// TwinCAT 3 PLC project SCADA_V2
// ProgramVersion: 3.1.4024.0
// libraries:
//   PlantControl and CMs, * (ArmAutomation)
//   Tc2_ControllerToolbox, * (Beckhoff Automation GmbH)
//   Tc2_Standard, * (Beckhoff Automation GmbH)
//   Tc2_System, * (Beckhoff Automation GmbH)
//   Tc3_Module, * (Beckhoff Automation GmbH)
// project tree:
//   GVLs/ CMD.TcGVL, HMI.TcGVL, GVL.TcGVL, PAR.TcGVL, SEQ.TcGVL, SIM.TcGVL
//   / PlcTask.TcTTO
//   POUs/CMs/ CM_AI_CALL.TcPOU, CM_DO_3state_CALL.TcPOU, CM_DO_CALL.TcPOU
//   POUs/EQ Modules/ EQ_CALL.TcPOU, EQ_Conveyor_V1.TcPOU
//   POUs/HVAC/ HVAC_B28_CM_CALL.TcPOU, HVAC_B28_Main_Seq.TcPOU
//   POUs/Plant Control/ FB_PlantControl_B57.TcPOU, FB_PlantControl_B28.TcPOU
//   POUs/Regulators/ PRG_FB_CTRL_PID.TcPOU, PRG_PID_CALL.TcPOU
//   POUs/ SITE_100MS.TcPOU, SITE_MAIN_CYCLIC.TcPOU
//   POUs/Simulations/ CALL_SIM.TcPOU, FBALT_2_PUMPS_GRAPH.TcPOU, FB_ALT_2_PUMPS.TcPOU, SIM_Analog_Input.TcPOU, SIM_Valve_Damper_OPEN_CLOSE.TcPOU
// real-time tasks:
//   TASK SITE_MAIN_CYCLIC: cycle T#10ms, priority 20, ADS port 350
//   TASK SITE_100MS: cycle T#100000us, priority 1, ADS port 351

CONFIGURATION SCADA_V2
    RESOURCE PLC ON TwinCAT3
        TASK PlcTask(INTERVAL := T#10ms, PRIORITY := 20);
        PROGRAM SITE_MAIN_CYCLIC WITH PlcTask : SITE_MAIN_CYCLIC;
        PROGRAM SITE_100MS WITH PlcTask : SITE_100MS;
    END_RESOURCE
END_CONFIGURATION

// ---- GVLs/CMD.TcGVL
{attribute 'qualified_only'}
VAR_GLOBAL
	Plant_B57_Control : PlantAndCMs.Udt_PlantControl;
	
	Plant_B28_Control : PlantAndCMs.Udt_PlantControl;
END_VAR

// ---- GVLs/HMI.TcGVL
{attribute 'qualified_only'}
VAR_GLOBAL
	
	//CMs for HVAC
	CM_AV_1 : PlantAndCMs.Udt_CM_Actuator2State_V2;
	
	CM_PU_AO_1 : PlantAndCMs.Udt_CM_AO_V2;
	
	CM_MTR_AO_1 : PlantAndCMs.Udt_CM_AO_V2;
	MTR_1_PO_PV : DINT;
	
	CM_DMP_AO_1 : PlantAndCMs.Udt_CM_Actuator2State_V2;
	
	//CMs For EQs
	CM_MTR_3State : PlantAndCMs.Udt_CM_Actuator3State_V2;

	//
	outputFromPressure_1 : LREAL;
	
	
	//PID
	CM_DMP_1_PID_PARAMS : ST_CTRL_PID_PARAMS;
	CM_MTR_1_PID_PARAMS : ST_CTRL_PID_PARAMS;
	
	//Simulation parameters
	
	
	
	
	
	//SP
	
	MTR_1_MAN_SP : DINT;
	DMP_1_MAN_SP : DINT;
	
END_VAR

// ---- GVLs/GVL.TcGVL
{attribute 'qualified_only'}
VAR_GLOBAL
	
	mb_Input_Coils    :    ARRAY [0..255] OF BOOL;
	mb_Output_Coils :    ARRAY [0..255] OF BOOL;
	mb_Input_Registers :    ARRAY [0..255] OF WORD; // Modbus TCP master side function code = 04 (read only)
	mb_Output_Registers :    ARRAY [0..255] OF WORD; // Modbus TCP master side function code = 03 & 16 (read/write)
	 
END_VAR

// ---- GVLs/PAR.TcGVL
{attribute 'qualified_only'}
VAR_GLOBAL
	
	// DAMPER SP
	
	DMP_1_SP : INT; 
	
	//Motor SP
	
	MTR_1_SP : DINT;

END_VAR

// ---- GVLs/SEQ.TcGVL
{attribute 'qualified_only'}
VAR_GLOBAL
	
	// HVAC_SEQ_28
	
	B28_STEP_1: BOOL;
	B28_STEP_2 : BOOL;
	B28_STEP_3 : BOOL;
	B28_STEP_4 : BOOL;
	B28_STEP_5 : BOOL;
	B28_STEP_6: BOOL;

END_VAR

// ---- GVLs/SIM.TcGVL
{attribute 'qualified_only'}
VAR_GLOBAL
	
	Pressure_1_Input : DINT;
	Pressure_1 : REAL ;
	
	//Sim Damper
	
	Feedback_Open : BOOL;
	Feedback_Closed : BOOL;
	
	DMP_1_INPUT : DINT;
	DMP_1_OUTPUT : DINT;
	
	MTR_1_InputFromPID : DINT;
	MTR_1_OutputToPID : DINT;
	
	// Conveyor sim
	
	CV_ON: BOOL;
	CCV_ON: BOOL;
	
END_VAR

// ---- POUs/SITE_MAIN_CYCLIC.TcPOU
PROGRAM SITE_MAIN_CYCLIC
VAR
	PlantControl_B57 : FB_PlantControl_B57;
	PlantControl_B28 : FB_PlantControl_B28;
	
	SIM_CALL : CALL_SIM;
	
	HVAC_CM_CALL : HVAC_B28_CM_CALL;
	
	HVAC_MAIN_SEQ : HVAC_B28_Main_Seq;
	
	cm_AI_CALL : CM_AI_CALL;
	cm_DO_3State_CALL : CM_DO_3state_CALL;
	
END_VAR

PlantControl_B28();
PlantControl_B57();


//B28
HVAC_CM_CALL();
HVAC_MAIN_SEQ();

//For testing:
EQ_CALL();
SIM_CALL();

// CMs
cm_AI_CALL();
//cm_DO_3State_CALL();

END_PROGRAM

// ---- POUs/Plant Control/FB_PlantControl_B57.TcPOU
FUNCTION_BLOCK FB_PlantControl_B57

VAR
	Plant_Control : PlantAndCMs.FB_PlantControl_V2;
	
	
	MB_START : BOOL;
	MB_EMG_STOP : BOOL;
END_VAR

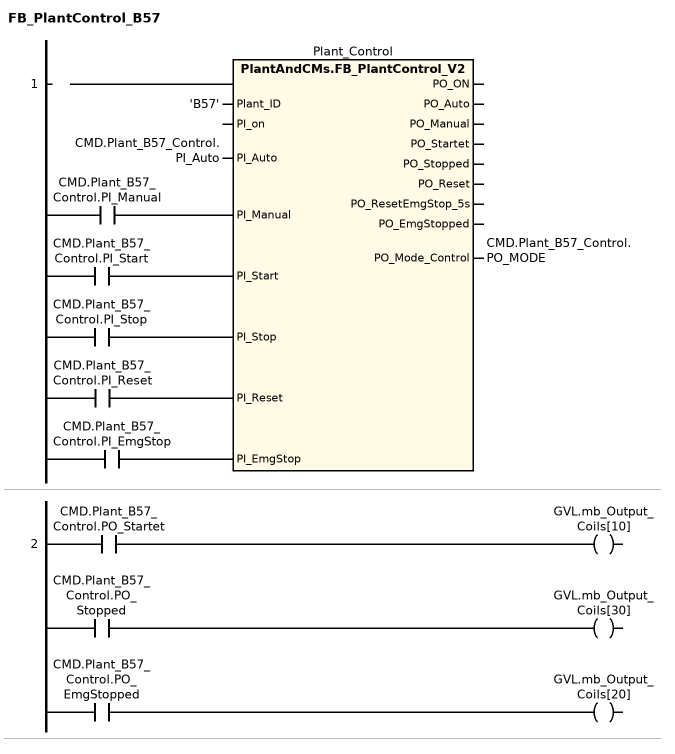
// NETWORK 1
Plant_Control(
    Plant_ID := 'B57',
    PI_Auto := CMD.Plant_B57_Control.PI_Auto,
    PI_Manual := CMD.Plant_B57_Control.PI_Manual,
    PI_Start := CMD.Plant_B57_Control.PI_Start,
    PI_Stop := CMD.Plant_B57_Control.PI_Stop,
    PI_Reset := CMD.Plant_B57_Control.PI_Reset,
    PI_EmgStop := CMD.Plant_B57_Control.PI_EmgStop,
    PO_Mode_Control => CMD.Plant_B57_Control.PO_MODE); // PlantAndCMs.FB_PlantControl_V2

// NETWORK 2
GVL.mb_Output_Coils[10] := CMD.Plant_B57_Control.PO_Startet;
GVL.mb_Output_Coils[30] := CMD.Plant_B57_Control.PO_Stopped;
GVL.mb_Output_Coils[20] := CMD.Plant_B57_Control.PO_EmgStopped;

END_FUNCTION_BLOCK

// ---- POUs/Plant Control/FB_PlantControl_B28.TcPOU
FUNCTION_BLOCK FB_PlantControl_B28

VAR
	Plant_Control : PlantAndCMs.FB_PlantControl_V2;
	
	
	MB_START : BOOL;
	MB_EMG_STOP : BOOL;
END_VAR

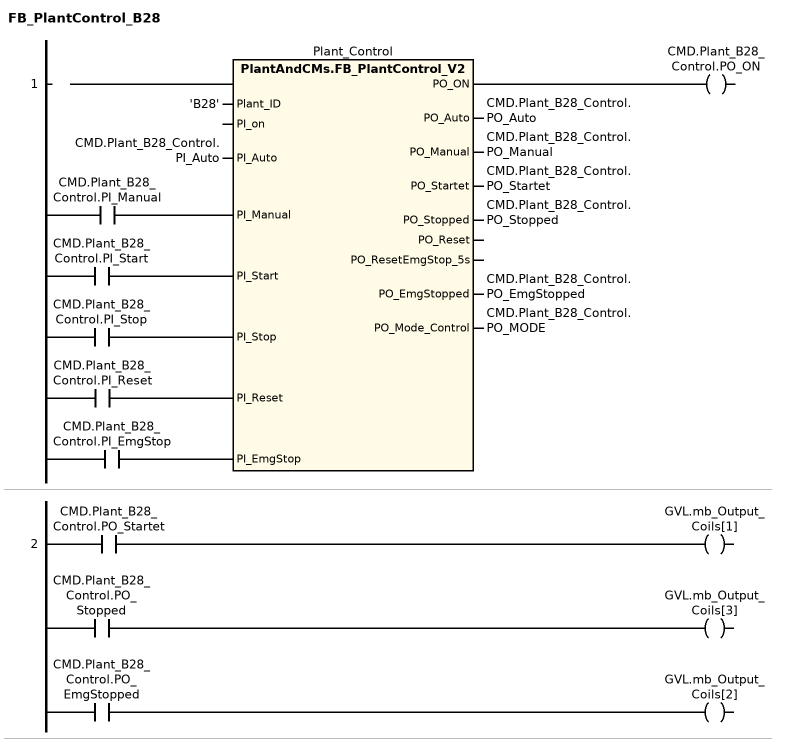
// NETWORK 1
Plant_Control(
    Plant_ID := 'B28',
    PI_Auto := CMD.Plant_B28_Control.PI_Auto,
    PI_Manual := CMD.Plant_B28_Control.PI_Manual,
    PI_Start := CMD.Plant_B28_Control.PI_Start,
    PI_Stop := CMD.Plant_B28_Control.PI_Stop,
    PI_Reset := CMD.Plant_B28_Control.PI_Reset,
    PI_EmgStop := CMD.Plant_B28_Control.PI_EmgStop,
    PO_Auto => CMD.Plant_B28_Control.PO_Auto,
    PO_Manual => CMD.Plant_B28_Control.PO_Manual,
    PO_Startet => CMD.Plant_B28_Control.PO_Startet,
    PO_Stopped => CMD.Plant_B28_Control.PO_Stopped,
    PO_EmgStopped => CMD.Plant_B28_Control.PO_EmgStopped,
    PO_Mode_Control => CMD.Plant_B28_Control.PO_MODE); // PlantAndCMs.FB_PlantControl_V2
CMD.Plant_B28_Control.PO_ON := Plant_Control.PO_ON;

// NETWORK 2
GVL.mb_Output_Coils[1] := CMD.Plant_B28_Control.PO_Startet;
GVL.mb_Output_Coils[3] := CMD.Plant_B28_Control.PO_Stopped;
GVL.mb_Output_Coils[2] := CMD.Plant_B28_Control.PO_EmgStopped;

END_FUNCTION_BLOCK

// ---- POUs/Simulations/CALL_SIM.TcPOU
FUNCTION_BLOCK CALL_SIM
VAR_INPUT
END_VAR
VAR_OUTPUT
END_VAR
VAR
	Damper_1_SIM : SIM_Valve_Damper_OPEN_CLOSE;
	
	pressure_1_SIM : SIM_Analog_Input;
	
	fb_ALT_2_PUMPS : FB_ALT_2_PUMPS;
	LS1:BOOL;
	LS2:BOOL;
	LS3:BOOL;
	LS4:BOOL;
	
	Pump_1 : BOOL;
	Pump_2 : BOOL;
	min_limit: INT;
END_VAR


IF SEQ.B28_STEP_2 THEN
	Damper_1_SIM(
	max_limit := PAR.DMP_1_SP,
	min_limit := 0,
	
	Start_Open := SEQ.B28_STEP_2,
	Start_Close := FALSE,//SEQ.B28_STEP_3,
	Open_Finish => SIM.Feedback_Open,
	Close_Finish => SIM.Feedback_Closed,
	open_status => SIM.DMP_1_OUTPUT
	
);
END_IF


fb_ALT_2_PUMPS(
	LS_1 := LS1,
	LS_2 := LS2,
	LS_3 := LS3,
	
	Pump_1 => Pump_1,
	Pump_2 => Pump_2
	);

pressure_1_SIM(
	EnableSim := CMD.Plant_B28_Control.PO_ON,
	AutoMode := SEQ.B28_STEP_3,
	ManualValue :=  HMI.MTR_1_MAN_SP,
	AutoSpeed := 0.1,
	MinValue := 15000,
	MaxValue := 30000,
	ManualValue := 10,
	SimulatedValue => SIM.Pressure_1,
	);

END_FUNCTION_BLOCK

// ---- POUs/Simulations/SIM_Valve_Damper_OPEN_CLOSE.TcPOU
FUNCTION_BLOCK SIM_Valve_Damper_OPEN_CLOSE
VAR_INPUT
    Start_Open  : BOOL;
    Start_Close : BOOL;
    max_limit   : INT;
    min_limit   : INT;
END_VAR

VAR_OUTPUT
    Open_Finish  : BOOL:= FALSE;
    Close_Finish : BOOL := FALSE;
    open_status  : INT := 0;
END_VAR

VAR
    timer : TON;
END_VAR

// Start timer only if movement is requested and not yet at limit
IF (Start_Open AND open_status < max_limit) OR (Start_Close AND open_status > min_limit) THEN
    timer(IN := TRUE, PT := T#1S);
ELSE
    timer(IN := FALSE);
END_IF

// On timer expiration, step open_status up or down
IF timer.Q THEN
    IF Start_Open AND open_status < max_limit THEN
        open_status := open_status + 1;
    ELSIF Start_Close AND open_status > min_limit THEN
        open_status := open_status - 1;
    END_IF
    timer(IN := FALSE); // Reset timer after action
END_IF

// Output flags
Open_Finish  := (open_status >= max_limit);
Close_Finish := (open_status <= min_limit);

END_FUNCTION_BLOCK

// ---- POUs/Simulations/SIM_Analog_Input.TcPOU
FUNCTION_BLOCK SIM_Analog_Input
VAR_INPUT
    EnableSim   : BOOL;
    AutoMode    : BOOL;
    ManualValue : REAL;
    AutoSpeed   : REAL;         // e.g. 0.1
    
	MinValue    : REAL;         // e.g. 0.0
    MaxValue    : REAL;         // e.g. 100.0
END_VAR

VAR_OUTPUT
    SimulatedValue : REAL;
END_VAR

VAR
    timeCounter : REAL := 0.0;
    timer       : TON;
END_VAR

// Auto simulation mode
IF EnableSim THEN
    IF AutoMode THEN
        timer(IN := TRUE, PT := T#500ms);
        IF timer.Q THEN
            timer(IN := FALSE); // reset
            timeCounter := timeCounter + AutoSpeed;
            SimulatedValue := (MaxValue - MinValue)/2.0 * SIN(timeCounter) + (MaxValue + MinValue)/2.0;
        END_IF
    ELSE
        // Manual override mode
        SimulatedValue := LIMIT(MinValue, ManualValue, MaxValue);
    END_IF
ELSE
    // Simulation disabled
    SimulatedValue := 0.0;
    timer(IN := FALSE);
END_IF

END_FUNCTION_BLOCK

// ---- POUs/Simulations/FB_ALT_2_PUMPS.TcPOU
FUNCTION_BLOCK FB_ALT_2_PUMPS
VAR_INPUT
	LS_1 : BOOL;
	LS_2 : BOOL;
	LS_3 : BOOL;
	LS_4 : BOOL;
END_VAR
VAR_OUTPUT
	Pump_1 : BOOL;
	Pump_2 : BOOL;
END_VAR
VAR
	Reset_pumps: BOOL;
	Alt_pumps: BOOL;
	
	Pump_Count : INT := 0;
	LS_2_Pump_1: BOOL;
	LS_2_Pump_2: BOOL;
	LS_3_Pump_1: BOOL;
	LS_3_Pump_2: BOOL;
END_VAR
VAR // added by the converter: edge detectors and wires of the graphical bodies
    _rt1 : R_TRIG;
    _w1, _w2, _w3 : BOOL;
END_VAR

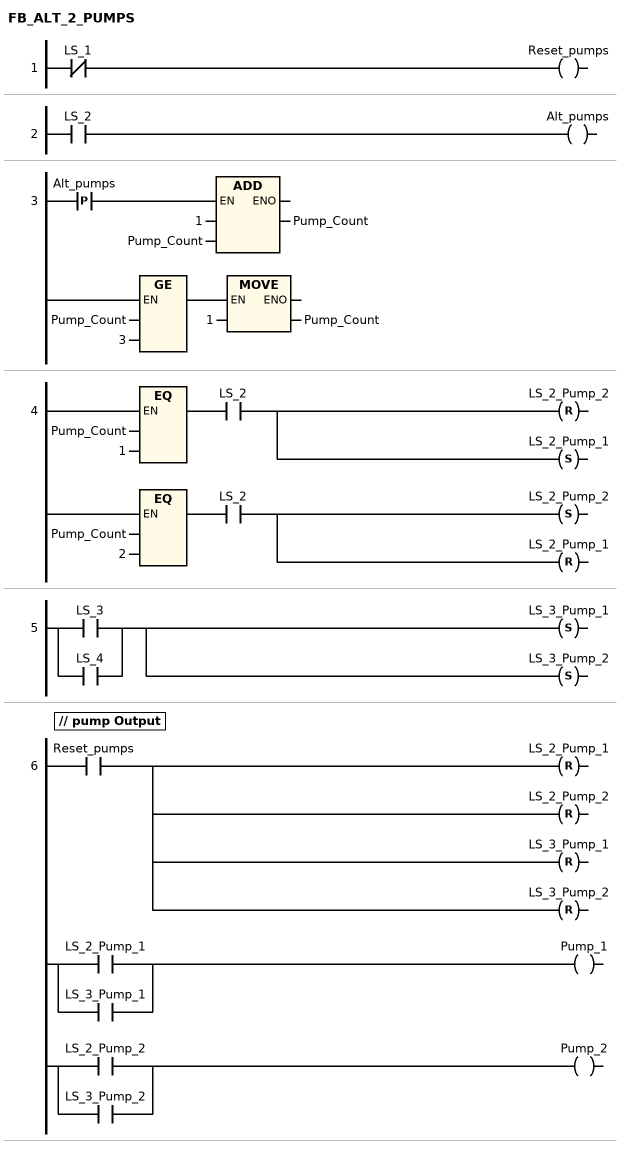
// NETWORK 1
Reset_pumps := NOT LS_1;

// NETWORK 2
Alt_pumps := LS_2;

// NETWORK 3
_rt1(CLK := Alt_pumps);
IF _rt1.Q THEN Pump_Count := 1 + Pump_Count; END_IF
IF Pump_Count >= 3 THEN Pump_Count := 1; END_IF

// NETWORK 4
_w1 := Pump_Count = 1 AND LS_2;
LS_2_Pump_2 R= _w1;
LS_2_Pump_1 S= _w1;
_w2 := Pump_Count = 2 AND LS_2;
LS_2_Pump_2 S= _w2;
LS_2_Pump_1 R= _w2;

// NETWORK 5
_w3 := LS_3 OR LS_4;
LS_3_Pump_1 S= _w3;
LS_3_Pump_2 S= _w3;

// NETWORK 6
// label: // pump Output
LS_2_Pump_1 R= Reset_pumps;
LS_2_Pump_2 R= Reset_pumps;
LS_3_Pump_1 R= Reset_pumps;
LS_3_Pump_2 R= Reset_pumps;
Pump_1 := LS_2_Pump_1 OR LS_3_Pump_1;
Pump_2 := LS_2_Pump_2 OR LS_3_Pump_2;

END_FUNCTION_BLOCK

// ---- POUs/HVAC/HVAC_B28_CM_CALL.TcPOU
FUNCTION_BLOCK HVAC_B28_CM_CALL
VAR_INPUT
END_VAR
VAR_OUTPUT
END_VAR
VAR
	AI_1_Temp : PlantAndCMs.CM_SensorAnalog_V2;
	AI_2_Pres: PlantAndCMs.CM_SensorAnalog_V2;
	
	AI_DMP_1: PlantAndCMs.CM_SensorAnalog_V2;
	
	AV_1 : PlantAndCMs.CM_Actuator2State_V2;
	AV_2 : PlantAndCMs.CM_Actuator2State_V2;
	
	MTR_1 : PlantAndCMs.CM_AO_V2;
	MTR_2 : PlantAndCMs.CM_AO_V2;
	
	DMP_1 : PlantAndCMs.CM_AO_V2;
	
	
	
	DMP_2 : PlantAndCMs.CM_AO_V2;
	
END_VAR

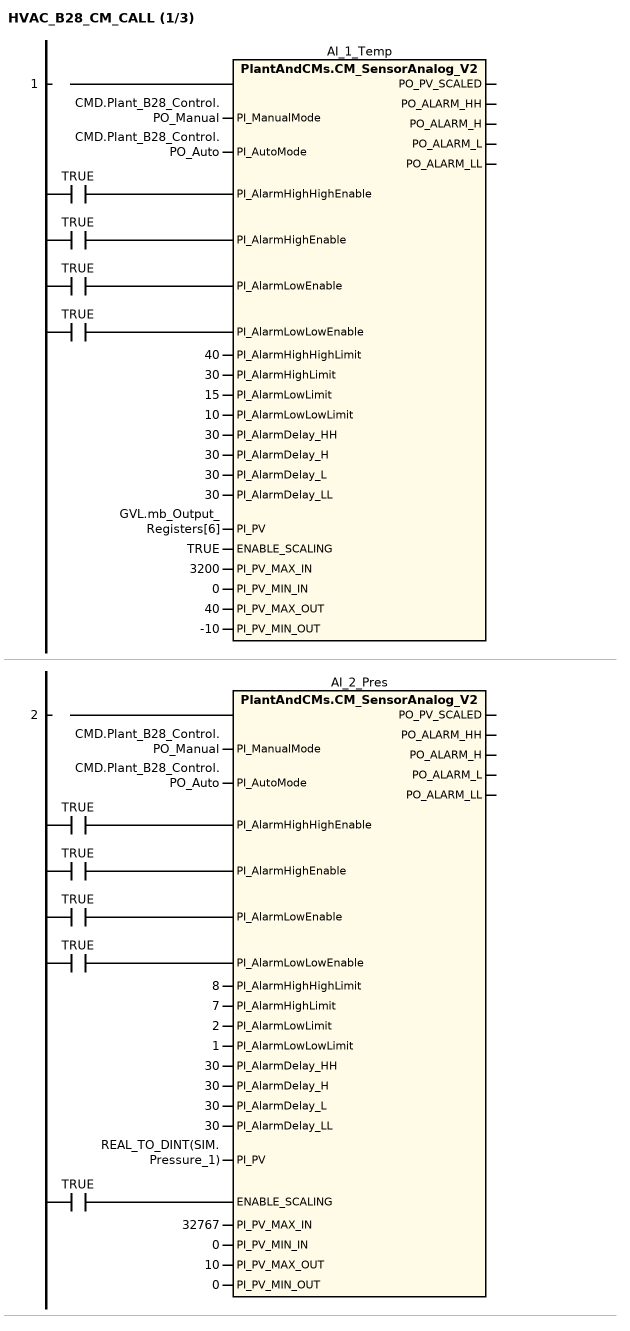
// NETWORK 1
AI_1_Temp(
    PI_ManualMode := CMD.Plant_B28_Control.PO_Manual,
    PI_AutoMode := CMD.Plant_B28_Control.PO_Auto,
    PI_AlarmHighHighEnable := TRUE,
    PI_AlarmHighEnable := TRUE,
    PI_AlarmLowEnable := TRUE,
    PI_AlarmLowLowEnable := TRUE,
    PI_AlarmHighHighLimit := 40,
    PI_AlarmHighLimit := 30,
    PI_AlarmLowLimit := 15,
    PI_AlarmLowLowLimit := 10,
    PI_AlarmDelay_HH := 30,
    PI_AlarmDelay_H := 30,
    PI_AlarmDelay_L := 30,
    PI_AlarmDelay_LL := 30,
    PI_PV := GVL.mb_Output_Registers[6],
    ENABLE_SCALING := TRUE,
    PI_PV_MAX_IN := 3200,
    PI_PV_MIN_IN := 0,
    PI_PV_MAX_OUT := 40,
    PI_PV_MIN_OUT := -10); // PlantAndCMs.CM_SensorAnalog_V2

// NETWORK 2
AI_2_Pres(
    PI_ManualMode := CMD.Plant_B28_Control.PO_Manual,
    PI_AutoMode := CMD.Plant_B28_Control.PO_Auto,
    PI_AlarmHighHighEnable := TRUE,
    PI_AlarmHighEnable := TRUE,
    PI_AlarmLowEnable := TRUE,
    PI_AlarmLowLowEnable := TRUE,
    PI_AlarmHighHighLimit := 8,
    PI_AlarmHighLimit := 7,
    PI_AlarmLowLimit := 2,
    PI_AlarmLowLowLimit := 1,
    PI_AlarmDelay_HH := 30,
    PI_AlarmDelay_H := 30,
    PI_AlarmDelay_L := 30,
    PI_AlarmDelay_LL := 30,
    PI_PV := REAL_TO_DINT(SIM.Pressure_1),
    ENABLE_SCALING := TRUE,
    PI_PV_MAX_IN := 32767,
    PI_PV_MIN_IN := 0,
    PI_PV_MAX_OUT := 10,
    PI_PV_MIN_OUT := 0); // PlantAndCMs.CM_SensorAnalog_V2

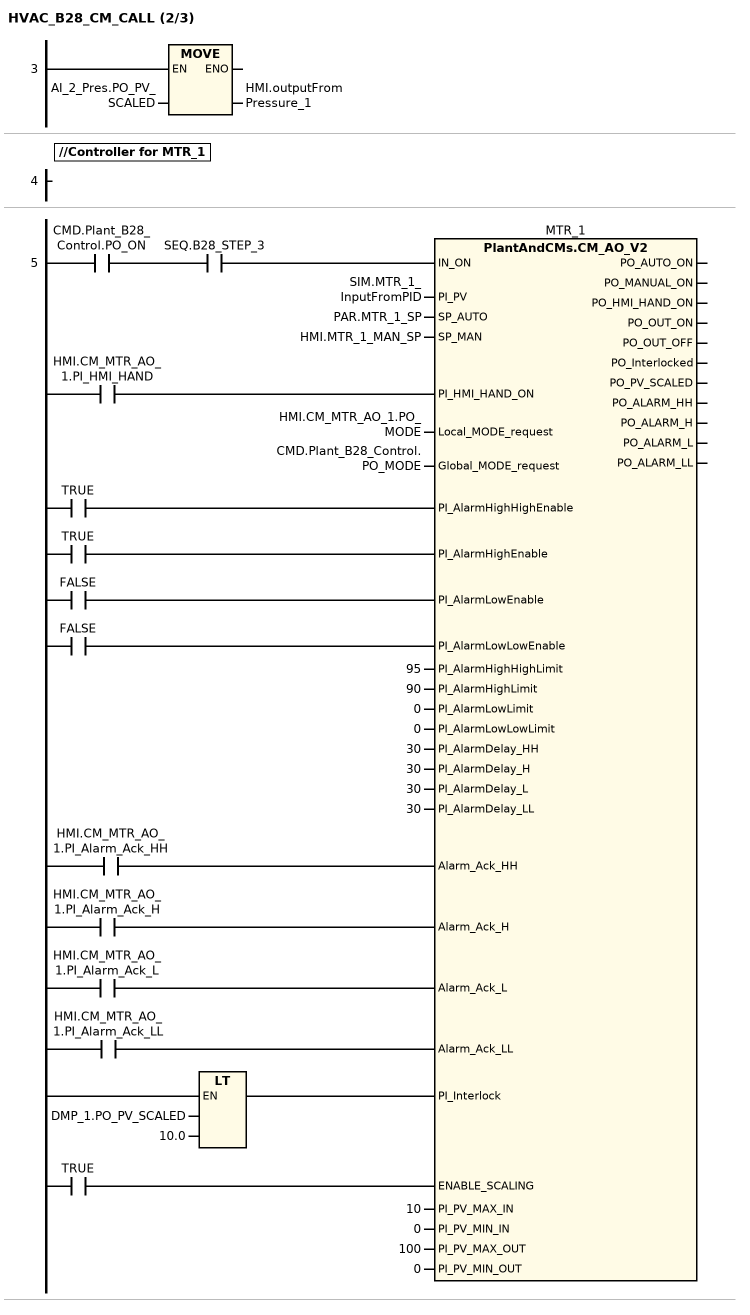
// NETWORK 3
HMI.outputFromPressure_1 := AI_2_Pres.PO_PV_SCALED;

// NETWORK 4
// label: //Controller for MTR_1

// NETWORK 5
MTR_1(
    IN_ON := CMD.Plant_B28_Control.PO_ON AND SEQ.B28_STEP_3,
    PI_PV := SIM.MTR_1_InputFromPID,
    SP_AUTO := PAR.MTR_1_SP,
    SP_MAN := HMI.MTR_1_MAN_SP,
    PI_HMI_HAND_ON := HMI.CM_MTR_AO_1.PI_HMI_HAND,
    Local_MODE_request := HMI.CM_MTR_AO_1.PO_MODE,
    Global_MODE_request := CMD.Plant_B28_Control.PO_MODE,
    PI_AlarmHighHighEnable := TRUE,
    PI_AlarmHighEnable := TRUE,
    PI_AlarmLowEnable := FALSE,
    PI_AlarmLowLowEnable := FALSE,
    PI_AlarmHighHighLimit := 95,
    PI_AlarmHighLimit := 90,
    PI_AlarmLowLimit := 0,
    PI_AlarmLowLowLimit := 0,
    PI_AlarmDelay_HH := 30,
    PI_AlarmDelay_H := 30,
    PI_AlarmDelay_L := 30,
    PI_AlarmDelay_LL := 30,
    Alarm_Ack_HH := HMI.CM_MTR_AO_1.PI_Alarm_Ack_HH,
    Alarm_Ack_H := HMI.CM_MTR_AO_1.PI_Alarm_Ack_H,
    Alarm_Ack_L := HMI.CM_MTR_AO_1.PI_Alarm_Ack_L,
    Alarm_Ack_LL := HMI.CM_MTR_AO_1.PI_Alarm_Ack_LL,
    PI_Interlock := DMP_1.PO_PV_SCALED < 10.0,
    ENABLE_SCALING := TRUE,
    PI_PV_MAX_IN := 10,
    PI_PV_MIN_IN := 0,
    PI_PV_MAX_OUT := 100,
    PI_PV_MIN_OUT := 0); // PlantAndCMs.CM_AO_V2

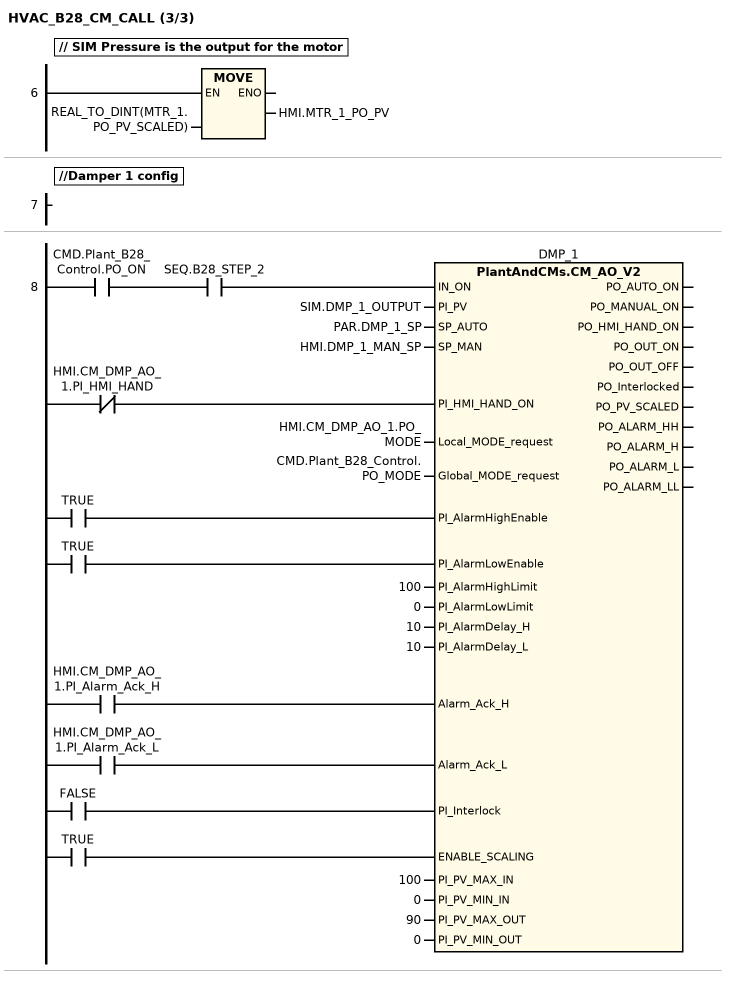
// NETWORK 6
// label: // SIM Pressure is the output for the motor
HMI.MTR_1_PO_PV := REAL_TO_DINT(MTR_1.PO_PV_SCALED);

// NETWORK 7
// label: //Damper 1 config

// NETWORK 8
DMP_1(
    IN_ON := CMD.Plant_B28_Control.PO_ON AND SEQ.B28_STEP_2,
    PI_PV := SIM.DMP_1_OUTPUT,
    SP_AUTO := PAR.DMP_1_SP,
    SP_MAN := HMI.DMP_1_MAN_SP,
    PI_HMI_HAND_ON := NOT HMI.CM_DMP_AO_1.PI_HMI_HAND,
    Local_MODE_request := HMI.CM_DMP_AO_1.PO_MODE,
    Global_MODE_request := CMD.Plant_B28_Control.PO_MODE,
    PI_AlarmHighEnable := TRUE,
    PI_AlarmLowEnable := TRUE,
    PI_AlarmHighLimit := 100,
    PI_AlarmLowLimit := 0,
    PI_AlarmDelay_H := 10,
    PI_AlarmDelay_L := 10,
    Alarm_Ack_H := HMI.CM_DMP_AO_1.PI_Alarm_Ack_H,
    Alarm_Ack_L := HMI.CM_DMP_AO_1.PI_Alarm_Ack_L,
    PI_Interlock := FALSE,
    ENABLE_SCALING := TRUE,
    PI_PV_MAX_IN := 100,
    PI_PV_MIN_IN := 0,
    PI_PV_MAX_OUT := 90,
    PI_PV_MIN_OUT := 0); // PlantAndCMs.CM_AO_V2

END_FUNCTION_BLOCK

// ---- POUs/HVAC/HVAC_B28_Main_Seq.TcPOU
FUNCTION_BLOCK HVAC_B28_Main_Seq
VAR_INPUT
END_VAR
VAR_OUTPUT
END_VAR
VAR
END_VAR

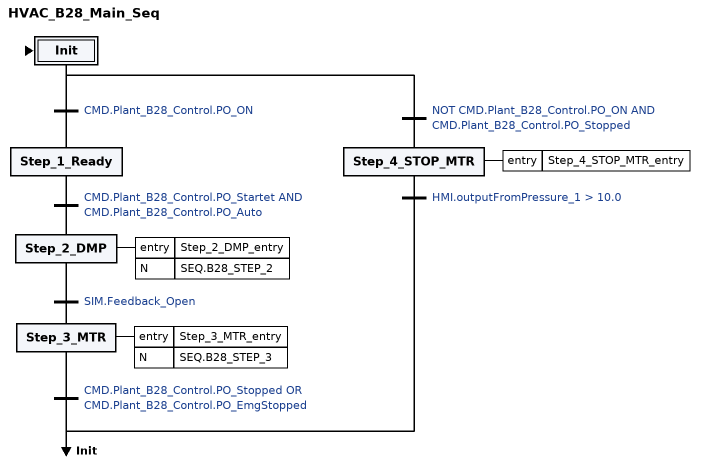
INITIAL_STEP Init:
END_STEP
TRANSITION FROM Init TO Step_1_Ready
    := CMD.Plant_B28_Control.PO_ON;
END_TRANSITION
STEP Step_1_Ready:
END_STEP
TRANSITION FROM Step_1_Ready TO Step_2_DMP
    := CMD.Plant_B28_Control.PO_Startet AND CMD.Plant_B28_Control.PO_Auto;
END_TRANSITION
STEP Step_2_DMP:
    Step_2_DMP_entry(P1);  // entry action
    SEQ.B28_STEP_2(N);
END_STEP
TRANSITION FROM Step_2_DMP TO Step_3_MTR
    := SIM.Feedback_Open;
END_TRANSITION
STEP Step_3_MTR:
    Step_3_MTR_entry(P1);  // entry action
    SEQ.B28_STEP_3(N);
END_STEP
TRANSITION FROM Step_3_MTR TO Init
    := CMD.Plant_B28_Control.PO_Stopped OR CMD.Plant_B28_Control.PO_EmgStopped;
END_TRANSITION
TRANSITION FROM Init TO Step_4_STOP_MTR
    := NOT CMD.Plant_B28_Control.PO_ON AND CMD.Plant_B28_Control.PO_Stopped;
END_TRANSITION
STEP Step_4_STOP_MTR:
    Step_4_STOP_MTR_entry(P1);  // entry action
END_STEP
TRANSITION FROM Step_4_STOP_MTR TO Init
    := HMI.outputFromPressure_1 > 10.0;
END_TRANSITION

ACTION Step_2_DMP_entry:
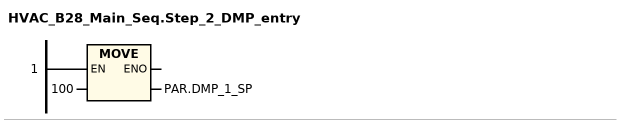
// NETWORK 1
PAR.DMP_1_SP := 100;
END_ACTION

ACTION Step_3_MTR_entry:
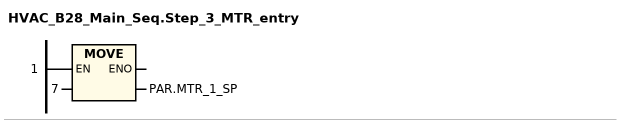
// NETWORK 1
PAR.MTR_1_SP := 7;
END_ACTION

ACTION Step_4_STOP_MTR_entry:
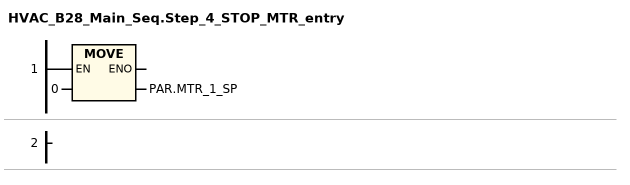
// NETWORK 1
PAR.MTR_1_SP := 0;

// NETWORK 2
END_ACTION

END_FUNCTION_BLOCK

// ---- POUs/CMs/CM_AI_CALL.TcPOU
FUNCTION_BLOCK CM_AI_CALL
VAR_INPUT
END_VAR
VAR_OUTPUT
END_VAR
VAR
END_VAR

// NETWORK 1

END_FUNCTION_BLOCK

// ---- POUs/CMs/CM_DO_3state_CALL.TcPOU
FUNCTION_BLOCK CM_DO_3state_CALL
VAR_INPUT
END_VAR
VAR_OUTPUT
END_VAR
VAR
	
END_VAR

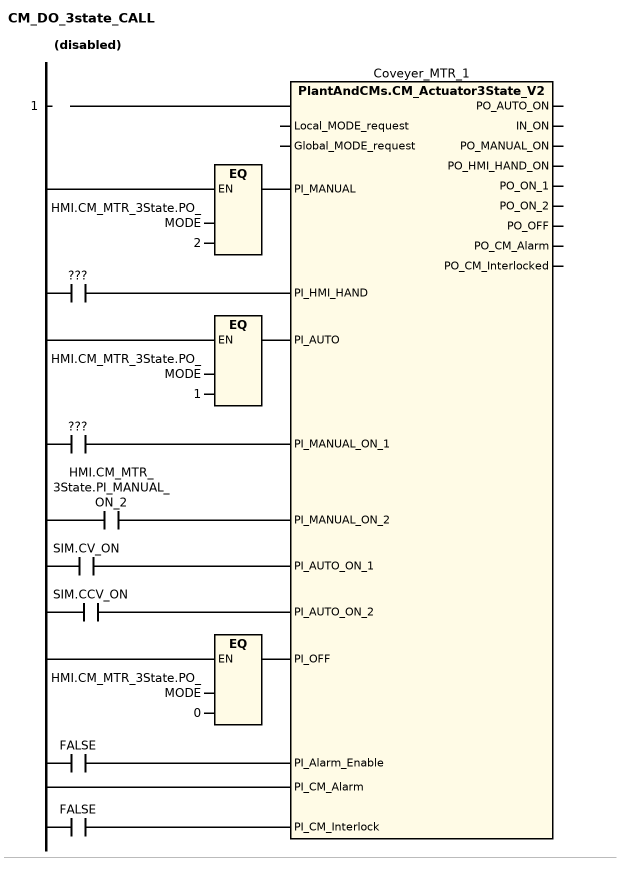
// NETWORK 1 (disabled)
// Coveyer_MTR_1(
//     PI_MANUAL := HMI.CM_MTR_3State.PO_MODE = 2,
//     PI_AUTO := HMI.CM_MTR_3State.PO_MODE = 1,
//     PI_MANUAL_ON_2 := HMI.CM_MTR_3State.PI_MANUAL_ON_2,
//     PI_AUTO_ON_1 := SIM.CV_ON,
//     PI_AUTO_ON_2 := SIM.CCV_ON,
//     PI_OFF := HMI.CM_MTR_3State.PO_MODE = 0,
//     PI_Alarm_Enable := FALSE,
//     PI_CM_Alarm := TRUE,
//     PI_CM_Interlock := FALSE); // PlantAndCMs.CM_Actuator3State_V2

END_FUNCTION_BLOCK

// ---- POUs/EQ Modules/EQ_CALL.TcPOU
PROGRAM EQ_CALL
VAR
	//EQ
	conveyor_V1 : EQ_Conveyor_V1;
	
	
	//CM
	Coveyer_MTR_1 : PlantAndCMs.CM_Actuator3State_V2;
END_VAR

conveyor_V1(	
				
				M_101_CW => SIM.CV_ON,
				M_101_CCW => SIM.CCV_ON
);

Coveyer_MTR_1(
	Local_MODE_request:= HMI.CM_MTR_3State.PO_MODE, 
	Global_MODE_request:= CMD.Plant_B28_Control.PO_MODE, 
	PI_MANUAL:= HMI.CM_MTR_3State.PO_MODE = 2, 
	PI_HMI_HAND:= Coveyer_MTR_1.PI_HMI_HAND, 
	PI_AUTO:= HMI.CM_MTR_3State.PO_MODE = 1 , 
	PI_MANUAL_ON_1:= Coveyer_MTR_1.PI_MANUAL_ON_1, 
	PI_MANUAL_ON_2:= Coveyer_MTR_1.PI_MANUAL_ON_2, 
	PI_AUTO_ON_1:= SIM.CV_ON, 
	PI_AUTO_ON_2:= SIM.CCV_ON, 
	PI_OFF:= HMI.CM_MTR_3State.PO_MODE = 0 , 
	PI_Alarm_Enable:= FALSE, 
	PI_CM_Alarm:= FALSE, 
	PI_CM_Interlock:= conveyor_V1.Alarm_1 OR conveyor_V1.Alarm_2, 
	IN_ON=> , 
	PO_AUTO_ON=> , 
	PO_MANUAL_ON=> , 
	PO_HMI_HAND_ON=> , 
	PO_ON_1=> , 
	PO_ON_2=> , 
	PO_OFF=> , 
	PO_CM_Alarm=> , 
	PO_CM_Interlocked=> 
	);

END_PROGRAM

// ---- POUs/EQ Modules/EQ_Conveyor_V1.TcPOU
FUNCTION_BLOCK EQ_Conveyor_V1
VAR_INPUT
	PS_101: BOOL; // Proximity switch
	PS_102: BOOL;
	
	STOP: BOOL;
END_VAR
VAR_OUTPUT
	M_101_CW : BOOL;
	M_101_CCW : BOOL;
	
	Alarm_1: BOOL;
	Alarm_2: BOOL;
END_VAR
VAR
	TRIG_LS_101: Tc2_Standard.R_TRIG;
	TRIG_LS_102: Tc2_Standard.R_TRIG;
	SR_M_101_CW: SR;
	SR_M_101_CCW: SR;
	TON_M101_CW: TON;
	TON_M102_CW: TON;
	
END_VAR

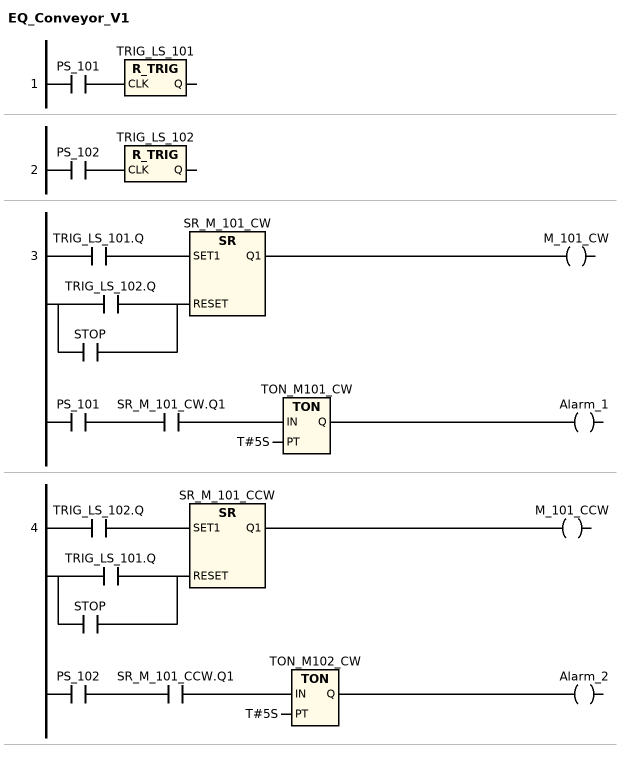
// NETWORK 1
TRIG_LS_101(CLK := PS_101); // R_TRIG

// NETWORK 2
TRIG_LS_102(CLK := PS_102); // R_TRIG

// NETWORK 3
SR_M_101_CW(SET1 := TRIG_LS_101.Q, RESET := TRIG_LS_102.Q OR STOP); // SR
M_101_CW := SR_M_101_CW.Q1;
TON_M101_CW(IN := PS_101 AND SR_M_101_CW.Q1, PT := T#5S); // TON
Alarm_1 := TON_M101_CW.Q;

// NETWORK 4
SR_M_101_CCW(SET1 := TRIG_LS_102.Q, RESET := TRIG_LS_101.Q OR STOP); // SR
M_101_CCW := SR_M_101_CCW.Q1;
TON_M102_CW(IN := PS_102 AND SR_M_101_CCW.Q1, PT := T#5S); // TON
Alarm_2 := TON_M102_CW.Q;

END_FUNCTION_BLOCK

// ---- POUs/SITE_100MS.TcPOU
PROGRAM SITE_100MS
VAR
	
END_VAR



PRG_PID_CALL();

END_PROGRAM

// ---- POUs/Regulators/PRG_PID_CALL.TcPOU
PROGRAM PRG_PID_CALL
VAR
	//B28
	B28_MTR_1_PID : PlantAndCMs.FB_PID;
	
	
END_VAR

(*
// MOTOR 1 PID CALL
HMI.CM_MTR_1_PID_PARAMS.tCtrlCycleTime := T#500MS;
HMI.CM_MTR_1_PID_PARAMS.tTaskCycleTime := T#100MS;
HMI.CM_MTR_1_PID_PARAMS.fKp := 5.0;	
HMI.CM_MTR_1_PID_PARAMS.tTd := T#500MS;
HMI.CM_MTR_1_PID_PARAMS.tTn := T#100S;
HMI.CM_MTR_1_PID_PARAMS.tTv := T#200MS;	
HMI.CM_MTR_1_PID_PARAMS.fOutMinLimit := 0.0;
HMI.CM_MTR_1_PID_PARAMS.fOutMaxLimit := 100.0;


B28_MTR_1_PID(
	IN_stCTRL_PID_PARAMS := HMI.CM_MTR_1_PID_PARAMS
	);

HMI.CM_DMP_1_PID_PARAMS.tCtrlCycleTime := T#500MS;
HMI.CM_DMP_1_PID_PARAMS.tTaskCycleTime := T#100MS;
HMI.CM_DMP_1_PID_PARAMS.fKp := 5.0;	
HMI.CM_DMP_1_PID_PARAMS.tTd := T#500MS;
HMI.CM_DMP_1_PID_PARAMS.tTn := T#100S;
HMI.CM_DMP_1_PID_PARAMS.tTv := T#200MS;	
HMI.CM_DMP_1_PID_PARAMS.fOutMinLimit := 0.0;
HMI.CM_DMP_1_PID_PARAMS.fOutMaxLimit := 180.0;

B28_DMP_1_PID(
	IN_stCTRL_PID_PARAMS := HMI.CM_MTR_1_PID_PARAMS
	);
*)

PRG_FB_CTRL_PID();

END_PROGRAM

// ---- POUs/Regulators/PRG_FB_CTRL_PID.TcPOU
PROGRAM PRG_FB_CTRL_PID
VAR
	fSetpointValue					: LREAL;
	fActualValue					: LREAL;
	fManSyncValue					: LREAL;
	bSync							: BOOL;

	fOut							: LREAL;
	bHold							: BOOL;

	eMode							: E_CTRL_MODE;
	stCTRL_PID_PARAMS				: ST_CTRL_PID_PARAMS;
	stCTRL_PID_PARAMS_MTR_1			: ST_CTRL_PID_PARAMS;

	eErrorId						: E_CTRL_ERRORCODES;
	bError							: BOOL;
	bARWactive						: BOOL;

	(* controllers *)
	fbCTRL_PID						: FB_CTRL_PID;
	fbCTRL_PID_B28_MTR_1			: FB_CTRL_PID;

	bInit							: BOOL	:= TRUE;
	bInit_MTR_1						: BOOL	:= TRUE;
	fbTON							: TON;
	
	
	
	
END_VAR


IF CMD.Plant_B28_Control.PO_MODE = 2 THEN
	eMode :=  4;	
END_IF
IF CMD.Plant_B28_Control.PO_MODE = 1  THEN
	eMode :=  2;
ELSE
	eMode :=  0;	
END_IF


IF bInit THEN
	(* init parameter struct *)
	stCTRL_PID_PARAMS.tCtrlCycleTime		:= T#500MS;	//used to control the actual sample time of the PID algorythm, must be = or > than the task cycle time
	stCTRL_PID_PARAMS.tTaskCycleTime		:= T#100MS;		// must be the same as the cycletime configured in the task which the regulator is called in (CyclicTask100Ms)
	stCTRL_PID_PARAMS.fKp					:= 5.0;			(* proportional gain Kp				*)
	stCTRL_PID_PARAMS.tTn					:= T#100S;		(*  Tn								*)
	stCTRL_PID_PARAMS.tTv					:= T#200MS;		(*  Tv								*)
	stCTRL_PID_PARAMS.tTd					:= T#500MS;		(*  Td								*)
	stCTRL_PID_PARAMS.fOutMaxLimit			:=  100.0;			(* maximum output limit			(for  fillValve)	*) 
	stCTRL_PID_PARAMS.fOutMinLimit			:= -0.0;			(* minimum output limit			(for  fillValve)	*)

	(* set the mode to ACTIVE --> normal operation *)
	eMode := eCTRL_MODE_ACTIVE;

	(* reset the init flag *)
	bInit := FALSE;
END_IF

IF bInit_MTR_1 THEN
	(* init parameter struct *)
	stCTRL_PID_PARAMS_MTR_1.tCtrlCycleTime		:= T#500MS;	//used to control the actual sample time of the PID algorythm, must be = or > than the task cycle time
	stCTRL_PID_PARAMS_MTR_1.tTaskCycleTime		:= T#100MS;		// must be the same as the cycletime configured in the task which the regulator is called in (CyclicTask100Ms)
	stCTRL_PID_PARAMS_MTR_1.fKp					:= 0.1;			(* proportional gain Kp				*)
	stCTRL_PID_PARAMS_MTR_1.tTn					:= T#100S;		(*  Tn								*)
	stCTRL_PID_PARAMS_MTR_1.tTv					:= T#100MS;		(*  Tv								*)
	stCTRL_PID_PARAMS_MTR_1.tTd					:= T#500MS;		(*  Td								*)
	stCTRL_PID_PARAMS_MTR_1.fOutMaxLimit			:=  100.0;			(* maximum output limit			(for  fillValve)	*) 
	stCTRL_PID_PARAMS_MTR_1.fOutMinLimit			:= -0.0;			(* minimum output limit			(for  fillValve)	*)

	(* set the mode to ACTIVE --> normal operation *)
	eMode := eCTRL_MODE_ACTIVE;

	(* reset the init flag *)
	bInit_MTR_1 := FALSE;
END_IF

(*
TYPE E_CTRL_MODE :
(
    eCTRL_MODE_IDLE       := 0, (* mode idle *)
    eCTRL_MODE_PASSIVE    := 1, (* mode passive *)
    eCTRL_MODE_ACTIVE     := 2, (* mode active *)
    eCTRL_MODE_RESET      := 3, (* mode reset *)
    eCTRL_MODE_MANUAL     := 4, (* mode manual *)
    eCTRL_MODE_TUNE       := 5, (* mode tuning *)
    eCTRL_MODE_SELFTEST       := 6, (* mode selftest *)
    eCTRL_MODE_SYNC_MOVEMENT  := 7  (* mode synchronize *)
);
END_TYPE
*)

(*
fActualValue :=  FIO.iPV; 	//FIO.rLevelMeter;
fSetpointValue := FIO.iSP; //FIO.rSetPoint (0-10V Scaled to 0-300 cm)

(* copy var to scope var *)
GVL.fSetpointValueToScope 	:= fSetpointValue;
GVL.fActualValueToScope 	:= fActualValue;
*)

(* call controller *)
fbCTRL_PID(		fSetpointValue		:= fSetpointValue,
				fActualValue		:= fActualValue, //feedback value (proces variable)
				fManSyncValue		:= fManSyncValue, // controll fOut directly with 0-100 %?
				bSync				:= bSync,
				eMode				:= eMode,
				bHold				:= bHold,
				stParams			:= stCTRL_PID_PARAMS,
				fOut				=> fOut, // output to PID
				bARWactive			=> bARWactive,
				eErrorId			=> eErrorId,
				bError				=> bError
				);

(*
(* copy var to scope var *)
GVL.fOutToScope := fOut;
FIO.rFillValve :=  fOut;

GVL.outputDischargeValve := fOut;

(********************************************* CALL MOTOR 1 ***********************************************)
*)
fActualValue :=  HMI.outputFromPressure_1; 	// Fra tryk sensor (0-32767 --> 0-100)
fSetpointValue := PAR.MTR_1_SP; //F



fbCTRL_PID_B28_MTR_1(
				fSetpointValue		:= fSetpointValue,
				fActualValue		:= fActualValue, //feedback value (proces variable)
				fManSyncValue		:= fManSyncValue, // controll fOut directly with 0-100 %?
				bSync				:= bSync,
				eMode				:= eMode,
				bHold				:= bHold,
				stParams			:= stCTRL_PID_PARAMS_MTR_1,
				fOut				=> fOut, // output to PID
				bARWactive			=> bARWactive,
				eErrorId			=> eErrorId,
				bError				=> bError
				);

SIM.MTR_1_InputFromPID := LREAL_TO_DINT(fOut);

END_PROGRAM

// ---- POUs/CMs/CM_DO_CALL.TcPOU
FUNCTION_BLOCK CM_DO_CALL
VAR_INPUT
END_VAR
VAR_OUTPUT
END_VAR
VAR
END_VAR

// NETWORK 1

END_FUNCTION_BLOCK

// ---- POUs/Simulations/FBALT_2_PUMPS_GRAPH.TcPOU
FUNCTION_BLOCK FBALT_2_PUMPS_GRAPH
VAR_INPUT
	LS_1 : BOOL;
	LS_2 : BOOL;
	LS_3 : BOOL;
	LS_4 : BOOL;
	
END_VAR
VAR_OUTPUT
END_VAR
VAR
END_VAR

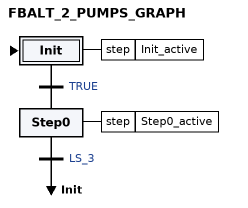
INITIAL_STEP Init:
    Init_active(N);  // step action
END_STEP
TRANSITION FROM Init TO Step0
    := TRUE;
END_TRANSITION
STEP Step0:
    Step0_active(N);  // step action
END_STEP
TRANSITION FROM Step0 TO Init
    := LS_3;
END_TRANSITION

ACTION Step0_active:
// NETWORK 1
END_ACTION

END_FUNCTION_BLOCK
